PROGRAM PRG_08_AnalogSignal
VAR
	uTurretValue: UDINT;
	iTRTEncoderValue: INT;
	TON_TeachLimit: TON;
	R_TRIG_TeachLimit: R_TRIG;
	RS_TurretBuffer: RS;
	R_TRIG_TurretBufferTrig: R_TRIG;
	F_TRIG_CarriageMedian: F_TRIG;
	TP_CarriageCaptureMedian: TP;
	F_TRIG_CarriageCaptureMedian: F_TRIG;
	F_TRIG_CarriageLeft: F_TRIG;
	TP_CarriageCaptureLeft: TP;
	F_TRIG_CarriageCaptureLeft: F_TRIG;
	F_TRIG_CarriageRight: F_TRIG;
	TP_CarriageCaptureRight: TP;
	F_TRIG_CarriageCaptureRight: F_TRIG;

	iCarriageAbsoluteMedian: INT;
	rCrossCutOffset: REAL;
	uCrossCutMax: UDINT;
	uCrossCutMin: UDINT;
	rRailHypotenuse: LREAL;
	iRailHypotenuse: UINT;
	uTeachLimit: UINT;
	rCarriageOffsetMultiplier: LREAL;
	rTurretOffsetMultiplier: LREAL;
	rCarriageVariable: LREAL;
	rTurretVariable: LREAL;
	iOffsetStep: INT;
	rCosineAngle: REAL;
	rConvertedOffset: REAL;
	iRailHypotenuseLeft: UINT;
	iRailHypotenuseRight: UINT;
	rAddend: REAL;
	R_TRIG_TurretValue: R_TRIG;
	
	bTurretEncoderCW: BOOL;
	bTurretEncoderCCW: BOOL;
	uTurretEncoderAddedValue: UDINT;
	
END_VAR

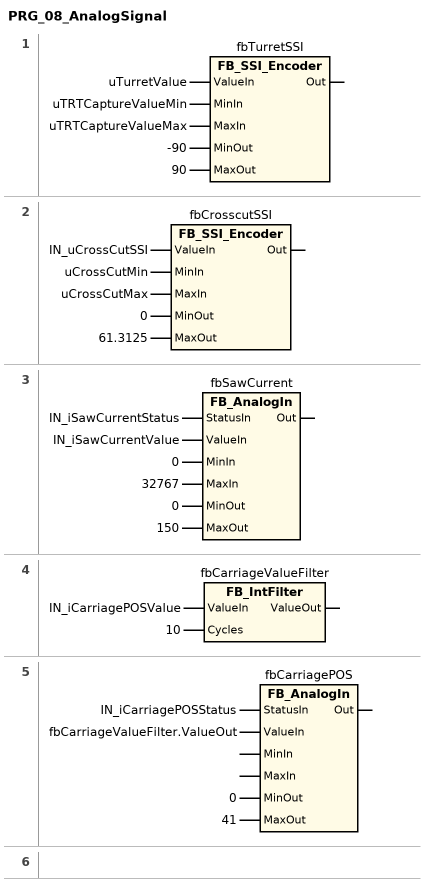
// NETWORK 1
fbTurretSSI(
    ValueIn := uTurretValue,
    MinIn := uTRTCaptureValueMin,
    MaxIn := uTRTCaptureValueMax,
    MinOut := -90,
    MaxOut := 90); // FB_SSI_Encoder

// NETWORK 2
fbCrosscutSSI(
    ValueIn := IN_uCrossCutSSI,
    MinIn := uCrossCutMin,
    MaxIn := uCrossCutMax,
    MinOut := 0,
    MaxOut := 61.3125); // FB_SSI_Encoder

// NETWORK 3
fbSawCurrent(
    StatusIn := IN_iSawCurrentStatus,
    ValueIn := IN_iSawCurrentValue,
    MinIn := 0,
    MaxIn := 32767,
    MinOut := 0,
    MaxOut := 150); // FB_AnalogIn

// NETWORK 4
fbCarriageValueFilter(ValueIn := IN_iCarriagePOSValue, Cycles := 10); // FB_IntFilter

// NETWORK 5
fbCarriagePOS(
    StatusIn := IN_iCarriagePOSStatus,
    ValueIn := fbCarriageValueFilter.ValueOut,
    MinOut := 0,
    MaxOut := 41); // FB_AnalogIn

// NETWORK 6

ACTION ACT_08_1_TurretSSI:
(* ########### ABSOLUTE 0 DEGREES: IN_uTurretSSI = 16238 @ SSI Data length of 15 ##################### *)
(* SSI Data length: 0x000F(15) *)

(* Turret Median, Max, Min *)
R_TRIG_TurretValue(CLK:= IN_bTurretRotationReference, Q=> );

	uTurretSSIMedian := 3188 + 32767 ;	// AP2 Turret median = 3188

	// Capture Min value and trigger stop at max CW
IF(* NOT *)IN_bTurretRotationReference AND (fbTurretSSI.Out.rScaled < -85) AND (IN_bTurretCW OR IN_bRemoteTrtCW) THEN
	uTRTCaptureValueMin := IN_uTurretSSI + 32767 - uTurretEncoderAddedValue ;		// Temp Min 21643
	bTurretMedian := FALSE ;
	bTurretCW := TRUE ;
	bTurretCCW := FALSE ;
	
	// Trigger stop at CW in case turret rotates past min value
ELSIF (uTRTCaptureValueMin <= uTRTCaptureValueMin - 50)	   THEN
	bTurretMedian := FALSE ;
	bTurretCW := TRUE ;
	bTurretCCW := FALSE ;

	// Capture Max value and trigger stop at max CCW
ELSIF ((* NOT *) IN_bTurretRotationReference AND (fbTurretSSI.Out.rScaled > 85) AND (IN_bTurretCCW OR IN_bRemoteTrtCCW)) OR
		((* NOT *) IN_bTurretRotationReference AND bTurretHome AND fbTurretSSI.Out.rScaled > 85) THEN
	uTRTCaptureValueMax := IN_uTurretSSI + 32767 - uTurretEncoderAddedValue ;		// Temp Max 50267
	bTurretMedian := FALSE ;
	bTurretCW := FALSE ;
	bTurretCCW := TRUE ;
	
	// Trigger stop at CCW in case turret rotates past max value
ELSIF (uTRTCaptureValueMax >= uTRTCaptureValueMax + 50)	  THEN
	bTurretMedian := FALSE ;
	bTurretCW := FALSE ;
	bTurretCCW := TRUE ;
	
	// Limits are off when Turret reference limit switch is triggered
ELSIF R_TRIG_TurretValue.Q AND  (fbTurretSSI.Out.rScaled > 85) THEN
	bTurretMedian := FALSE ;
	bTurretCW := FALSE ;
	bTurretCCW := FALSE ;
	
	// Limits are off when Turret reference limit switch is triggered
ELSIF R_TRIG_TurretValue.Q AND  (fbTurretSSI.Out.rScaled < -85) THEN
	bTurretMedian := FALSE ;
	bTurretCW := FALSE ;
	bTurretCCW := FALSE ;
	
END_IF

(* Turret rollover range *)		(* clockwise rollover, encoder value going down *)
IF ((IN_uTurretSSI <= 32767) AND (IN_uTurretSSI >= 20500)) THEN		// ########### dependent on range of encoder rollover #######################
	bTurretEncoderCW := TRUE ;
	uTurretEncoderAddedValue := 32767 ;
ELSE
	bTurretEncoderCW   := FALSE ;
	uTurretEncoderAddedValue := 0 ;
END_IF

(* Turret value going past min and max *)
IF (IN_uTurretSSI + 32767 - uTurretEncoderAddedValue < uTRTCaptureValueMax) AND (IN_uTurretSSI + 32767 - uTurretEncoderAddedValue > uTRTCaptureValueMin) THEN
	uTurretValue := IN_uTurretSSI + 32767 - uTurretEncoderAddedValue ;	
ELSIF (IN_uTurretSSI + 32767 - uTurretEncoderAddedValue > uTRTCaptureValueMax) THEN
	uTurretValue := uTRTCaptureValueMax ;
ELSIF (IN_uTurretSSI + 32767 - uTurretEncoderAddedValue < uTRTCaptureValueMin) THEN
	uTurretValue := uTRTCaptureValueMin ;
END_IF

(* Trigger stop turret at 0° *)
IF (IN_uTurretSSI + 32767 - uTurretEncoderAddedValue >= (uTurretSSIMedian-1)) AND (IN_uTurretSSI + 32767 - uTurretEncoderAddedValue <= (uTurretSSIMedian+1)) THEN
	bTurretMedianRange := TRUE;
ELSE bTurretMedianRange := FALSE;
END_IF 

(* ######################### NEW ############################# *)
(* Turret 0° - 45° range *)
IF fbTurretSSI.Out.rScaled > -47 AND fbTurretSSI.Out.rScaled < 47 THEN
	bTurret045Range := TRUE ;
ELSE bTurret045Range := FALSE ;
END_IF
(* ######################### NEW ############################# *)

(* Turret Encoder Display *)
(* (ValueIN/MaxIN)*32767  *)
OUT_iEncoderDisplay := iTRTEncoderValue ;
iTRTEncoderValue := REAL_TO_INT((((UDINT_TO_REAL(IN_uTurretSSI + 32767 - uTurretEncoderAddedValue - uTRTCaptureValueMin)) / UDINT_TO_REAL(uTRTCaptureValueMax - uTRTCaptureValueMin))*32767 ));
IF ((iTRTEncoderValue < 0) AND bTurretOverMedian) OR ((IN_uTurretSSI + 32767 - uTurretEncoderAddedValue > uTRTCaptureValueMax) AND bTurretOverMedian) THEN
	iTRTEncoderValue := 32767 ;
ELSIF ((iTRTEncoderValue < 0) AND bTurretUnderMedian) OR ((IN_uTurretSSI + 32767 - uTurretEncoderAddedValue < uTRTCaptureValueMin) AND bTurretUnderMedian) THEN
	iTRTEncoderValue := 0 ;
END_IF

(* Turret Return variable *)
IF (IN_uTurretSSI + 32767 - uTurretEncoderAddedValue > uTurretSSIMedian) AND NOT bTurretMedianRange THEN
	bTurretOverMedian := TRUE;
ELSE 	bTurretOverMedian := FALSE;
END_IF

IF (IN_uTurretSSI + 32767 - uTurretEncoderAddedValue < uTurretSSIMedian) AND NOT bTurretMedianRange THEN
	bTurretUnderMedian := TRUE;
ELSE 	bTurretUnderMedian := FALSE;
END_IF

(* Buffer zone for turret to slow down before approaching the trigger points at 0°, 90°, and -90° *)
R_TRIG_TurretBufferTrig(CLK:= bTurretMedianRange, Q=> );
RS_TurretBuffer(SET:= R_TRIG_TurretBufferTrig.Q, 
				RESET1:=  (IN_bTurretCCW OR IN_bRemoteTrtCCW OR IN_bTurretCW OR IN_bRemoteTrtCW), 
				Q1=> );

IF ((IN_uTurretSSI + 32767 - uTurretEncoderAddedValue >= (uTurretSSIMedian-100)) AND NOT (IN_uTurretSSI + 32767 - uTurretEncoderAddedValue >= uTurretSSIMedian) AND (IN_bTurretCCW OR IN_bRemoteTrtCCW OR (bTurretReturn AND OUT_bTrtCrgLH))) OR
	((IN_uTurretSSI + 32767 - uTurretEncoderAddedValue <= (uTurretSSIMedian+100)) AND NOT (IN_uTurretSSI + 32767 - uTurretEncoderAddedValue <= uTurretSSIMedian) AND (IN_bTurretCW OR IN_bRemoteTrtCW OR (bTurretReturn AND OUT_bTrtCrgRH))) OR
	((IN_uTurretSSI + 32767 - uTurretEncoderAddedValue <= (uTRTCaptureValueMin+100)) AND (IN_bTurretCW OR IN_bRemoteTrtCW OR (bTurretReturn AND OUT_bTrtCrgRH) OR bMachineHoming)) OR
	((IN_uTurretSSI + 32767 - uTurretEncoderAddedValue >= (uTRTCaptureValueMax-100)) AND (IN_bTurretCCW OR IN_bRemoteTrtCCW OR (bTurretReturn AND OUT_bTrtCrgLH) OR bMachineHoming))
THEN
	bTurretBufferSpeed := TRUE;
ELSE
	bTurretBufferSpeed := FALSE;
END_IF
END_ACTION

ACTION ACT_08_2_CrossCutSSI:
(* SSI Data length: 0x000F(15) *)
(* encoder values *)
uRailLimitLeft := 16210 ;//3746 ;	// align centre of the blade with the left inner edge of the bed rails
uRailLimitRight := 14953 ;//2625 ;	// align centre of the blade with the right inner edge of the bed rails
uCrossCutMax := 16356 ;//3893 ;		// move the saw block all the way to the left
uCrossCutMin := 15099 ;//2480 ;		// move the saw block all the way to the right

(* CrossCut Limits *)
IF (IN_uCrossCutSSI+32767 <= (uCrossCutMedian - (iRailHypotenuse - uTeachLimit))+32767) OR
	(((fbTurretSSI.Out.rScaled > 85 (*Degrees*)) OR (fbTurretSSI.Out.rScaled < -85)) AND (fbCrosscutSSI.Out.rScaled <= (fbCrosscutSSI.MinOut + 6 (*Inches*)))) OR
	(IN_uCrossCutSSI < (uCrossCutMin + 2))
	THEN
	bLimitRight := TRUE ;
	bLimitLeft := FALSE ;
ELSIF (IN_uCrossCutSSI+32767 >= (uCrossCutMedian + (iRailHypotenuse - uTeachLimit))+32767) OR
	(((fbTurretSSI.Out.rScaled > 85 (*Degrees*)) OR (fbTurretSSI.Out.rScaled < -85)) AND (fbCrosscutSSI.Out.rScaled >= (fbCrosscutSSI.MaxOut - 6 (*Inches*)))) OR
	(IN_uCrossCutSSI > (uCrossCutMax - 2))
	THEN
	bLimitLeft := TRUE ;
	bLimitRight := FALSE ;
ELSE
	bLimitRight := FALSE ;
	bLimitLeft 	:= FALSE ;
END_IF

(* Approaching Limits for Crosscut buffer zone *)
IF (IN_uCrossCutSSI+32767 <= (uCrossCutMedian - (iRailHypotenuse - uTeachLimit))+50+32767) OR 
	(((fbTurretSSI.Out.rScaled > 85 (*Degrees*)) OR (fbTurretSSI.Out.rScaled < -85)) AND (fbCrosscutSSI.Out.rScaled <= (fbCrosscutSSI.MinOut + 6)+1)) OR
	(IN_uCrossCutSSI <= (uCrossCutMin + 50))
	THEN
	bApproachingLimitRight := TRUE ;
	bApproachingLimitLeft := FALSE ;
ELSIF (IN_uCrossCutSSI+32767 >= (uCrossCutMedian + (iRailHypotenuse - uTeachLimit))-50+32767) OR 
	(((fbTurretSSI.Out.rScaled > 85 (*Degrees*)) OR (fbTurretSSI.Out.rScaled < -85)) AND (fbCrosscutSSI.Out.rScaled >= (fbCrosscutSSI.MaxOut - 6)-1))  OR
	(IN_uCrossCutSSI >= (uCrossCutMax - 50))
	THEN
	bApproachingLimitLeft := TRUE ;
	bApproachingLimitRight := FALSE ;
ELSE
	bApproachingLimitRight := FALSE ;
	bApproachingLimitLeft 	:= FALSE ;
END_IF

(*	bApproachingLimitRight := FALSE ;
	bApproachingLimitLeft 	:= FALSE ;
	bLimitRight := FALSE ;
	bLimitLeft 	:= FALSE ;
*)
(* Hypotenuse calculation *)
IF ABS(fbTurretSSI.Out.rScaled) <> 90 THEN
	rCosineAngle := COS ( (PI / 180) * ABS( fbTurretSSI.Out.rScaled)) ;
ELSE
	rCosineAngle := COS ( (PI / 180) * 89.9999 ) ;
END_IF

uTeachLimit := REAL_TO_UINT(((UDINT_TO_REAL(uRailLimitLeft - uRailLimitRight))/2) - ((UDINT_TO_REAL(uTeachLimitLeft - uTeachLimitRight))/2)) ;

fbTurretSSI.Out.rScaled ; // Turret Angle

	rRailHypotenuse := ( (UDINT_TO_LREAL(uRailLimitLeft - uRailLimitRight)/2) / rCosineAngle);
	
//	iRailHypotenuse := LREAL_TO_UINT(rRailHypotenuse);
IF rRailHypotenuse >= 6436 OR rRailHypotenuse < 0 THEN
	iRailHypotenuse := 6436;		// rRailHypotenuse = 6436 	@ 85°
ELSE
	iRailHypotenuse := LREAL_TO_UINT(rRailHypotenuse);
END_IF

(* Carriage Position Offset *)
fbCarriagePOS.Out.rScaled;
fbCrosscutSSI.Out.rScaled;

F_TRIG_CarriageMedian(CLK:= IN_bCarriageReference, Q=> );
TP_CarriageCaptureMedian(IN:= F_TRIG_CarriageMedian.Q, PT:= T#0.5S, Q=> , ET=> );
F_TRIG_CarriageCaptureMedian(CLK:= TP_CarriageCaptureMedian.Q, Q=> );
IF F_TRIG_CarriageCaptureMedian.Q THEN		
	iCarriageMedian := fbCarriageValueFilter.ValueOut ;
END_IF

iOffsetStep;
IF NOT IN_bCarriageReference THEN
	rCrossCutOffset := 0 ;
ELSE
	rCrossCutOffset := ABS(fbCarriagePOS.Out.rScaled - ((fbCarriagePOS.MaxOut-fbCarriagePOS.MinOut)/2)) + rAddend ;
		IF 		IN_bCarriageReference AND NOT bTurretMedianRange AND (fbCarriageValueFilter.ValueOut < iCarriageMedian AND fbTurretSSI.Out.rScaled > 55) THEN
			rAddend := 0.75 ; iOffsetStep := 1;	// Carriage left, Turret CCW
		ELSIF	IN_bCarriageReference AND NOT bTurretMedianRange AND (fbCarriageValueFilter.ValueOut > iCarriageMedian AND fbTurretSSI.Out.rScaled > 55) THEN
			rAddend := 0 ; iOffsetStep := 2;	// Carriage right, Turret CCW
		ELSIF	IN_bCarriageReference AND NOT bTurretMedianRange AND (fbCarriageValueFilter.ValueOut > iCarriageMedian AND fbTurretSSI.Out.rScaled < -55) THEN
			rAddend := 0.5 ; iOffsetStep := 3;	// Carriage right, Turret CW
		ELSIF	IN_bCarriageReference AND NOT bTurretMedianRange AND (fbCarriageValueFilter.ValueOut < iCarriageMedian AND fbTurretSSI.Out.rScaled < -55) THEN
			rAddend := 0 ; iOffsetStep := 4;	// Carriage left, Turret CW
		ELSE
			rAddend := 0 ; iOffsetStep := 10;
		END_IF
END_IF

(* Crosscut median *)
rTurretOffsetMultiplier := (rTurretVariable * (ABS(fbTurretSSI.Out.rScaled)/90)) ;

IF (NOT IN_bCarriageReference AND fbTurretSSI.Out.rScaled >0) OR (IN_bCarriageReference AND (fbTurretSSI.Out.rScaled > 85 OR fbTurretSSI.Out.rScaled < -85)) THEN	
	uCrossCutMedian := REAL_TO_UDINT (((UDINT_TO_REAL(uTeachLimitLeft + uTeachLimitRight)) / 2 ) -  ((rTurretOffsetMultiplier/(fbCrosscutSSI.MaxOut-fbCrosscutSSI.MinOut))*UDINT_TO_REAL(uCrossCutMax-uCrossCutMin))  ) ;
	rTurretVariable := 0.5;
ELSIF (NOT IN_bCarriageReference AND fbTurretSSI.Out.rScaled <0) OR (IN_bCarriageReference AND (fbTurretSSI.Out.rScaled > 85 OR fbTurretSSI.Out.rScaled < -85)) THEN	
	uCrossCutMedian := REAL_TO_UDINT (((UDINT_TO_REAL(uTeachLimitLeft + uTeachLimitRight)) / 2 ) +  ((rTurretOffsetMultiplier/(fbCrosscutSSI.MaxOut-fbCrosscutSSI.MinOut))*UDINT_TO_REAL(uCrossCutMax-uCrossCutMin))  ) ;
	rTurretVariable := 0.5;
ELSIF IN_bCarriageReference AND (fbCarriageValueFilter.ValueOut < iCarriageMedian) AND NOT (fbTurretSSI.Out.rScaled > 85 OR fbTurretSSI.Out.rScaled < -85) THEN
	uCrossCutMedian := REAL_TO_UDINT(((UDINT_TO_REAL(uTeachLimitLeft + uTeachLimitRight)) / 2 ) - ((rCrossCutOffset/(fbCrosscutSSI.MaxOut-fbCrosscutSSI.MinOut))*UDINT_TO_REAL(uCrossCutMax-uCrossCutMin)) /rCosineAngle) ;
ELSIF IN_bCarriageReference AND (fbCarriageValueFilter.ValueOut > iCarriageMedian) AND NOT (fbTurretSSI.Out.rScaled > 85 OR fbTurretSSI.Out.rScaled < -85) THEN
	uCrossCutMedian := REAL_TO_UDINT(((UDINT_TO_REAL(uTeachLimitLeft + uTeachLimitRight)) / 2 ) + ((rCrossCutOffset/(fbCrosscutSSI.MaxOut-fbCrosscutSSI.MinOut))*UDINT_TO_REAL(uCrossCutMax-uCrossCutMin)) /rCosineAngle) ;
END_IF

IF (IN_uCrossCutSSI >= (uCrossCutMedian - 10)) AND (IN_uCrossCutSSI <= (uCrossCutMedian + 10)) THEN
	bCrossCutCentre := TRUE ;
ELSE
	bCrossCutCentre := FALSE ;
END_IF
(* ################################################# REMOVE AFTER SETUP ########################
IF (IN_uCrossCutSSI >= (uCrossCutMedian - 30)) AND (IN_uCrossCutSSI <= (uCrossCutMedian + 30)) THEN
	bCrossCutCentreForRotation := TRUE ;
ELSE
	bCrossCutCentreForRotation := FALSE ;
END_IF
################################################# REMOVE AFTER SETUP ######################## *)
	bCrossCutCentreForRotation := TRUE ;

(* Teach Limits left and right *)
TON_TeachLimit(IN:= (IN_bTeach AND ((IN_bTeachLeft AND IN_uCrossCutSSI > (uCrossCutMedian+100)) OR (IN_bTeachRight AND IN_uCrossCutSSI < (uCrossCutMedian-100))) AND NOT IN_bCarriageReference AND bTurretMedianRange AND NOT (bTurretReturn OR bAutoCrossCut OR bMachineHoming OR OUT_bSawON)),
				PT:= T#3S, Q=> , ET=> );
OUT_bTeachLED := NOT TON_TeachLimit.Q AND IN_bTeach AND NOT IN_bCarriageReference AND bTurretMedianRange AND ((IN_bTeachLeft AND IN_uCrossCutSSI > (uCrossCutMedian+100)) OR (IN_bTeachRight AND IN_uCrossCutSSI < (uCrossCutMedian-100))) ;
R_TRIG_TeachLimit(CLK:= TON_TeachLimit.Q, Q=> );

IF NOT IN_bCarriageReference AND R_TRIG_TeachLimit.Q AND IN_bTeachLeft AND bTurretMedianRange AND NOT (bTurretReturn AND bAutoCrossCut AND bMachineHoming) THEN
	uTeachLimitLeft := IN_uCrossCutSSI;
ELSIF NOT IN_bCarriageReference AND R_TRIG_TeachLimit.Q AND IN_bTeachRight AND bTurretMedianRange AND NOT (bTurretReturn AND bAutoCrossCut AND bMachineHoming) THEN
	uTeachLimitRight := IN_uCrossCutSSI;
END_IF

(* crash positions *)
IF 		(fbCarriagePOS.Out.rScaled <= 24 AND fbTurretSSI.Out.rScaled >= 50 AND fbCrosscutSSI.Out.rScaled >= 46) 	// echain @ corner #1
	OR 	(fbCarriagePOS.Out.rScaled <= 41 AND fbTurretSSI.Out.rScaled >= 70 AND fbCrosscutSSI.Out.rScaled >= 57)		// light bar @ side 1-2
	OR	(fbCarriagePOS.Out.rScaled <= 30 AND fbTurretSSI.Out.rScaled <= -65 AND fbCrosscutSSI.Out.rScaled >= 59)	// corner 4
	OR	(fbCarriagePOS.Out.rScaled <= 30 AND fbTurretSSI.Out.rScaled >= 60 AND fbCrosscutSSI.Out.rScaled >= 51)		// echain @ corner #1
	OR	(fbCarriagePOS.Out.rScaled >= 36 AND fbTurretSSI.Out.rScaled <= -60 AND fbCrosscutSSI.Out.rScaled >= 60)	// corner 4
	OR	(fbCarriagePOS.Out.rScaled >= 30 AND fbTurretSSI.Out.rScaled <= -50 AND fbCrosscutSSI.Out.rScaled >= 57.5)	// corner 4
THEN
	bEchainCrashPosLeft := TRUE ;		// Crosscut Left limit
	bEchainCrashPosRight := FALSE ;
ELSIF 	(fbCarriagePOS.Out.rScaled <= 14 AND fbTurretSSI.Out.rScaled <= -85 AND fbCrosscutSSI.Out.rScaled <= 15) 	// echain @ corner #1
	OR	(fbCarriagePOS.Out.rScaled <= 17.5 AND fbTurretSSI.Out.rScaled >= 75 AND fbCrosscutSSI.Out.rScaled <= 10.5)	// echain @ corner #3
	OR  (fbCarriagePOS.Out.rScaled <= 30 AND fbTurretSSI.Out.rScaled <= -65 AND fbCrosscutSSI.Out.rScaled <= 7)		// light bar @ side 1-2
	OR  (fbCarriagePOS.Out.rScaled <= 10 AND fbTurretSSI.Out.rScaled <= -70 AND fbCrosscutSSI.Out.rScaled <= 16)	// echain @ corner #1
	OR  (fbCarriagePOS.Out.rScaled >= 21 AND fbTurretSSI.Out.rScaled >= 60 AND fbCrosscutSSI.Out.rScaled <= 7)		// corner #4
	OR  (fbCarriagePOS.Out.rScaled <= 21 AND fbTurretSSI.Out.rScaled >= 60 AND fbCrosscutSSI.Out.rScaled <= 7)		// servomotor side #3-4
	OR  (fbCarriagePOS.Out.rScaled <= 16 AND fbTurretSSI.Out.rScaled >= 60 AND fbCrosscutSSI.Out.rScaled <= 17)		// horizontal echain @ corner #3
	OR  (fbCarriagePOS.Out.rScaled >= 16 AND fbTurretSSI.Out.rScaled >= 65 AND fbCrosscutSSI.Out.rScaled <= 5)		// spray bar side #3-4
THEN
	bEchainCrashPosLeft := FALSE ;		// Crosscut Right limit
	bEchainCrashPosRight := TRUE ;
ELSE
	bEchainCrashPosLeft := FALSE ;
	bEchainCrashPosRight := FALSE ;
END_IF
END_ACTION

ACTION ACT_08_3_CarriagePOS:
(* Carriage end limits *)
F_TRIG_CarriageLeft(CLK:= IN_bCarriageLHLimit, Q=> );
TP_CarriageCaptureLeft(IN:= F_TRIG_CarriageLeft.Q, PT:= T#0.5S, Q=> , ET=> );
F_TRIG_CarriageCaptureLeft(CLK:= TP_CarriageCaptureLeft.Q, Q=> );
IF F_TRIG_CarriageCaptureLeft.Q THEN
	iCarriageLeftLimit := fbCarriageValueFilter.ValueOut ;
END_IF

IF fbCarriageValueFilter.ValueOut >= iCarriageLeftLimit THEN
	fbCarriagePOS.MinIn := iCarriageLeftLimit ;
ELSIF fbCarriageValueFilter.ValueOut < iCarriageLeftLimit THEN
	fbCarriagePOS.MinIn := fbCarriageValueFilter.ValueOut ;
END_IF


F_TRIG_CarriageRight(CLK:= IN_bCarriageRHLimit, Q=> );
TP_CarriageCaptureRight(IN:= F_TRIG_CarriageRight.Q, PT:= T#0.5S, Q=> , ET=> );
F_TRIG_CarriageCaptureRight(CLK:= TP_CarriageCaptureRight.Q, Q=> );
IF F_TRIG_CarriageCaptureRight.Q THEN
	iCarriageRightLimit := fbCarriageValueFilter.ValueOut ;
END_IF

IF fbCarriageValueFilter.ValueOut <= iCarriageRightLimit THEN
	fbCarriagePOS.MaxIn := iCarriageRightLimit ;
ELSIF fbCarriageValueFilter.ValueOut > iCarriageRightLimit THEN
	fbCarriagePOS.MaxIn := fbCarriageValueFilter.ValueOut ;
END_IF

iCarriageAbsoluteMedian := ( iCarriageRightLimit + iCarriageLeftLimit ) / 2 ;
END_ACTION

END_PROGRAM

(* stored: Version 1.1.0.1, ProductVersion 3.1.4024.12
   POU PRG_08_AnalogSignal: Id {08194954-8482-4d0c-916f-7e9a099a59da}, SpecialFunc None
   Action ACT_08_1_TurretSSI: Id {716da273-ea5c-4ef9-a865-fc5cb558ec9f}
   Action ACT_08_2_CrossCutSSI: Id {ac304cda-40d2-4e5a-8e98-9d9a7d6b6640}
   Action ACT_08_3_CarriagePOS: Id {524fab2b-6806-4c5b-acfa-b7a3368ebfbf} *)
